INTERFACE ITcoSafetySignals

{attribute 'monitoring' := 'call'}
PROPERTY AllKeysAuto : BOOL
GET
END_GET
END_PROPERTY

{attribute 'monitoring' := 'call'}
PROPERTY AllKeysNormal : BOOL
GET
END_GET
END_PROPERTY

{attribute 'monitoring' := 'call'}
PROPERTY AnyDeadman : BOOL
GET
END_GET
END_PROPERTY

{attribute 'monitoring' := 'call'}
PROPERTY AnyKeyManual : BOOL
GET
END_GET
END_PROPERTY

{attribute 'monitoring' := 'call'}
PROPERTY AnyKeyService : BOOL
GET
END_GET
END_PROPERTY

{attribute 'monitoring' := 'call'}
PROPERTY AnyKeyStep : BOOL
GET
END_GET
END_PROPERTY

{attribute 'monitoring' := 'call'}
PROPERTY IsAirPressureOk : BOOL
GET
END_GET
END_PROPERTY

{attribute 'monitoring' := 'call'}
PROPERTY IsDoorsOk : BOOL
GET
END_GET
END_PROPERTY

{attribute 'monitoring' := 'call'}
PROPERTY IsEstopOk : BOOL
GET
END_GET
END_PROPERTY

{attribute 'monitoring' := 'call'}
PROPERTY IsGlobalVoltageOK : BOOL
GET
END_GET
END_PROPERTY

{attribute 'monitoring' := 'call'}
PROPERTY IsLocalVoltageOk : BOOL
GET
END_GET
END_PROPERTY

END_INTERFACE

(* stored: Version 1.1.0.1
   Itf ITcoSafetySignals: Id {09f09e0c-75b1-4347-bd74-974be1821d01}
   Property AllKeysAuto: Id {abebcd61-9d16-4680-908c-879298cb6197}
   Get Get: Id {0c9c7b75-1873-4ee1-819e-5f0b90269d55}
   Property AllKeysNormal: Id {d67bac49-e277-48c2-ba54-9c1e54add6b8}
   Get Get: Id {e51a74eb-37af-47f8-8f4c-d46e69d3c0d3}
   Property AnyDeadman: Id {574e36d1-762a-4029-a603-3a970f29e339}
   Get Get: Id {edd3bdaa-e636-44bb-abc8-3717b9ba566a}
   Property AnyKeyManual: Id {69eb2418-3091-4c47-9298-e0655b8180cc}
   Get Get: Id {9870cbe0-67b8-4bae-9160-9bef87100de0}
   Property AnyKeyService: Id {6c11b35b-039e-471d-98c8-7ab7ebe51841}
   Get Get: Id {791d0b2f-c96c-4443-bdc5-c2f954507d49}
   Property AnyKeyStep: Id {46cfefee-aa6d-4e96-a445-d5aae557ccc0}
   Get Get: Id {0af6154d-7bc2-47b5-980a-4cf332211bc3}
   Property IsAirPressureOk: Id {8dcb80a2-2114-46bf-abaa-a96f6892b8a0}
   Get Get: Id {770c1924-2f84-40e4-93e0-573d766b1d10}
   Property IsDoorsOk: Id {63564c8d-5970-4f09-b7fa-3fd04fc00fc7}
   Get Get: Id {46b334ee-47df-4170-9548-f108c3b74678}
   Property IsEstopOk: Id {fef9d1c2-10a4-4048-b1ba-8414e00b6ed0}
   Get Get: Id {ec5d71a1-2551-4369-89d1-54b5709b2f35}
   Property IsGlobalVoltageOK: Id {d857c7ff-c99d-41ea-b8c1-648945fda4b4}
   Get Get: Id {392c5000-48b0-4616-8ded-e8e7a2dc1bc8}
   Property IsLocalVoltageOk: Id {a842c2ea-2c91-482e-9cfc-14a2150aba5a}
   Get Get: Id {ae6de065-b0e0-4efd-89d9-950dfa483ff8} *)
